{attribute 'c++_compatible'}
FUNCTION_BLOCK JsonSaxHandler IMPLEMENTS ITcJsonSaxHandler
VAR_INPUT
END_VAR
VAR_OUTPUT
END_VAR
VAR
	(* Values from JSON - written by callback methods *)	  
	sTimestamp 			: STRING(255);
	Sensor1				: LREAL;
	Sensor2				: DINT;
	
	(* State machine variables *)
	eState				: E_JsonStates;
	
	(* Indicators if an expected property has been found in JSON *)
	bStartObjectFound 	: BOOL;
	bEndObjectFound		: BOOL;
	bValuesFound 		: BOOL;
	bTimestampFound 	: BOOL;
	bTimestampValueFound: BOOL;
	bSensor1Found 		: BOOL;
	bSensor1ValueFound	: BOOL;
	bSensor2Found 		: BOOL;
	bSensor2ValueFound	: BOOL;
	
	(* Error indicators *)
	bError				: BOOL;
	sErrorMsg			: STRING(255);
END_VAR

IF bError THEN
	sErrorMsg := 'JSON message does not equal expected format';
END_IF

{attribute 'show'}
{attribute 'c++_compatible'}
{attribute 'minimal_input_size' := '4'}
{attribute 'pack_mode' := '4'}
{warning 'add method implementation'}
METHOD OnBool : HRESULT
VAR_INPUT
	value	: BOOL;
END_VAR
END_METHOD

{attribute 'show'}
{attribute 'c++_compatible'}
{attribute 'minimal_input_size' := '4'}
{attribute 'pack_mode' := '4'}
{warning 'add method implementation'}
METHOD OnDint : HRESULT
VAR_INPUT
	value	: DINT;
END_VAR
Sensor2 := value;
END_METHOD

{attribute 'show'}
{attribute 'c++_compatible'}
{attribute 'minimal_input_size' := '4'}
{attribute 'pack_mode' := '4'}
{warning 'add method implementation'}
METHOD OnEndArray : HRESULT
VAR_INPUT
	elementCount	: UDINT;
END_VAR
END_METHOD

{attribute 'show'}
{attribute 'c++_compatible'}
{attribute 'minimal_input_size' := '4'}
{attribute 'pack_mode' := '4'}
{warning 'add method implementation'}
METHOD OnEndObject : HRESULT
VAR_INPUT
	memberCount	: UDINT;
END_VAR
IF (eState = 100) THEN
	bEndObjectFound := TRUE;
	eState := 110;  
	ELSE
		IF (eState = 110) THEN
			bEndObjectFound := TRUE;
			eState := 120;
		ELSE
			bError := TRUE;  
	  END_IF			
END_IF
END_METHOD

{attribute 'show'}
{attribute 'c++_compatible'}
{attribute 'minimal_input_size' := '4'}
{attribute 'pack_mode' := '4'}
{warning 'add method implementation'}
METHOD OnKey : HRESULT
VAR_IN_OUT CONSTANT
	key	: STRING;
END_VAR
VAR_INPUT
	len	: UDINT;
END_VAR
IF ((eState = 20)AND(key = 'Values')) THEN
	bValuesFound := TRUE;
	eState := 30;
	ELSE
		IF ((eState = 40)AND(key = 'Timestamp')) THEN
		  bTimestampFound := TRUE;
		  eState := 50;
		ELSE
			IF ((eState = 60)AND(key = 'Sensor1')) THEN
				bSensor1Found := TRUE;
				eState := 70;
			ELSE
				IF ((eState = 80)AND(key = 'Sensor2')) THEN
					bSensor2Found := TRUE;
					eState := 90;
				ELSE
					bError := TRUE;
					Onkey := S_FALSE;
				END_IF				  
			END_IF	  
	  	END_IF
END_IF
END_METHOD

{attribute 'show'}
{attribute 'c++_compatible'}
{attribute 'minimal_input_size' := '4'}
{attribute 'pack_mode' := '4'}
{warning 'add method implementation'}
METHOD OnLint : HRESULT
VAR_INPUT
	value	: LINT;
END_VAR
END_METHOD

{attribute 'show'}
{attribute 'c++_compatible'}
{attribute 'minimal_input_size' := '4'}
{attribute 'pack_mode' := '4'}
{warning 'add method implementation'}
METHOD OnLreal : HRESULT
VAR_INPUT
	value	: LREAL;
END_VAR
IF (eState = 70) THEN
	bSensor1ValueFound := TRUE;
	Sensor1 := value;
	eState := 80;
ELSE
	bError := TRUE;
	OnLreal := S_FALSE;
END_IF
END_METHOD

{attribute 'show'}
{attribute 'c++_compatible'}
{attribute 'minimal_input_size' := '4'}
{attribute 'pack_mode' := '4'}
{warning 'add method implementation'}
METHOD OnNull : HRESULT
END_METHOD

{attribute 'show'}
{attribute 'c++_compatible'}
{attribute 'minimal_input_size' := '4'}
{attribute 'pack_mode' := '4'}
{warning 'add method implementation'}
METHOD OnRawNumber : HRESULT
VAR_IN_OUT CONSTANT
	value	: STRING;
END_VAR
VAR_INPUT
	len	: UDINT;
END_VAR
END_METHOD

{attribute 'show'}
{attribute 'c++_compatible'}
{attribute 'minimal_input_size' := '4'}
{attribute 'pack_mode' := '4'}
{warning 'add method implementation'}
METHOD OnStartArray : HRESULT
END_METHOD

{attribute 'show'}
{attribute 'c++_compatible'}
{attribute 'minimal_input_size' := '4'}
{attribute 'pack_mode' := '4'}
{warning 'add method implementation'}
METHOD OnStartObject : HRESULT
IF (eState = 10) THEN
	bStartObjectFound := TRUE;
	eState := 20;  
	ELSE
		IF (eState = 30) THEN
			bStartObjectFound := TRUE;
			eState := 40;
		ELSE
			bError := TRUE;  
	  END_IF			
END_IF
END_METHOD

{attribute 'show'}
{attribute 'c++_compatible'}
{attribute 'minimal_input_size' := '4'}
{attribute 'pack_mode' := '4'}
{warning 'add method implementation'}
METHOD OnString : HRESULT
VAR_IN_OUT CONSTANT
	value	: STRING;
END_VAR
VAR_INPUT
	len	: UDINT;
END_VAR
IF (eState = 50) THEN
	bTimestampValueFound := TRUE;
	STRNCPY(pDst:=ADR(sTimestamp), pSrc:=ADR(value), nDstSize:=SIZEOF(sTimestamp));
	eState := 60;
ELSE
	bError := TRUE;
	OnString := S_FALSE;
END_IF
END_METHOD

{attribute 'show'}
{attribute 'c++_compatible'}
{attribute 'minimal_input_size' := '4'}
{attribute 'pack_mode' := '4'}
{warning 'add method implementation'}
METHOD OnUdint : HRESULT
VAR_INPUT
	value	: UDINT;
END_VAR
IF (eState = 90) THEN
	bSensor2ValueFound := TRUE;
	Sensor2 := value;
	eState := 100;
ELSE
	bError := TRUE;
	OnUdint := S_FALSE;
END_IF
END_METHOD

{attribute 'show'}
{attribute 'c++_compatible'}
{attribute 'minimal_input_size' := '4'}
{attribute 'pack_mode' := '4'}
{warning 'add method implementation'}
METHOD OnUlint : HRESULT
VAR_INPUT
	value	: ULINT;
END_VAR
END_METHOD

{attribute 'show'}
{attribute 'c++_compatible'}
{attribute 'minimal_input_size' := '4'}
{attribute 'pack_mode' := '4'}
{warning 'add method implementation'}
METHOD TcAddRef : UDINT
END_METHOD

{attribute 'show'}
{attribute 'c++_compatible'}
{attribute 'minimal_input_size' := '4'}
{attribute 'pack_mode' := '4'}
{warning 'add method implementation'}
METHOD TcQueryInterface : HRESULT
VAR_INPUT
	iid	: REFERENCE TO IID;
	pipItf	: POINTER TO PVOID;
END_VAR
END_METHOD

{attribute 'show'}
{attribute 'c++_compatible'}
{attribute 'minimal_input_size' := '4'}
{attribute 'pack_mode' := '4'}
{warning 'add method implementation'}
METHOD TcRelease : UDINT
END_METHOD

END_FUNCTION_BLOCK

(* stored: Version 1.1.0.1, ProductVersion 3.1.4021.12
   POU JsonSaxHandler: Id {fd22ba04-0d36-44e7-a81e-c59d3ac0f333}, SpecialFunc None
   Method OnBool: Id {13455f88-e234-4d6f-b163-c3ace2d01de9}
   Method OnDint: Id {24238a66-3ba2-41ea-bb1d-dec022507274}
   Method OnEndArray: Id {1739a2d6-6bf1-4ae8-9382-66870451d46e}
   Method OnEndObject: Id {885811d0-5c76-4031-96ce-48dd447f7032}
   Method OnKey: Id {0166f13e-7ed0-43f7-a777-b23d02f1dd47}
   Method OnLint: Id {729de20b-2d3e-4125-9187-e0252a19c186}
   Method OnLreal: Id {e458c372-d873-4613-adb7-f607191d076c}
   Method OnNull: Id {65642340-6997-4108-83d9-c8813a05825e}
   Method OnRawNumber: Id {f9737890-9bac-4333-b9b2-37d74169c053}
   Method OnStartArray: Id {655fbaa9-4596-43be-8c13-3d5daaf75b5e}
   Method OnStartObject: Id {9da87a42-4b27-47bf-b4fc-3d1a5b5e45be}
   Method OnString: Id {1c13bada-871d-4b30-bee1-08ea70607c6f}
   Method OnUdint: Id {296ac94a-f1f7-4890-a4b8-5d9fd3b55ce6}
   Method OnUlint: Id {3d01b1c5-c02d-481b-a604-269325783bc9}
   Method TcAddRef: Id {ed9db009-45ee-459b-bd3c-e6eebd2276ca}
   Method TcQueryInterface: Id {bf125ab6-3d6a-4df3-b162-942f3b1feb6f}
   Method TcRelease: Id {f07919cf-792d-4887-afc7-1c9d1066ed11} *)
